{attribute 'Tc2GvlVarNames'}
VAR_GLOBAL
	Dem_Serrage_Presseurs_Manu,
	Dem_Desserrage_Presseurs_Manu					:BOOL;
	
	Dem_Serrage_Presseur_Amont_Laser_Auto,
	Dem_Desserrage_Presseur_Amont_Laser_Auto,
	Dem_Serrage_Presseur_Aval_Laser_Auto,
	Dem_Desserrage_Presseur_Aval_Laser_Auto			:BOOL;                                          	
	                                            		
	Distance_Annulation_Presseur_Laser				:LREAL;//Pnc_Presseurs
	Offset_Position_Desserree_Presseurs_Laser		:LREAL:=310;//Distance du tas où on considère le presseur assez relevé, correspond à la capcité max VP-300- + sécu arbitraire
	Def_Calib_Presseurs								:BOOL;	//Si problème pendant le calibrage, par exemple le preseur bloqué et ne descend pas tout en bas ou encore si descente sur profil
END_VAR

(* stored: Version 1.1.0.1, ProductVersion 3.1.4024.15
   GVL Global_Var_Presseurs_Laser: Id {52dd2bcc-2609-4b94-a13f-d70167a56370} *)
